FUNCTION_BLOCK FB_PanelDetect
VAR_INPUT
END_VAR
VAR_OUTPUT
END_VAR
VAR
	m_panelOnCounts :INT :=0;
	m_panelOnCountThres :INT :=50;
END_VAR

// check if panel is on
METHOD run : BOOL
VAR_INPUT
	IOValue :UDINT;
END_VAR
//Panel single  At installation--2#0000   not installation --2#0101
IF (IOValue AND 16#06) = 0 THEN
	m_panelOnCounts := MIN( m_panelOnCounts +1,m_panelOnCountThres);
ELSIF (IOValue AND 16#06) = 6  THEN
	m_panelOnCounts :=0;
END_IF
run := m_panelOnCounts >= m_panelOnCountThres;
END_METHOD

END_FUNCTION_BLOCK

(* stored: Version 1.1.0.1, ProductVersion 3.1.4024.11
   POU FB_PanelDetect: Id {47cf5248-c8cb-4b89-a8d5-96d08d2b209c}, SpecialFunc None
   Method run: Id {b2b5e204-adc8-4a47-b4a0-7ccab0ad6803} *)
